{attribute addProperty BoxType "EP7342-0002-0021"}
{attribute addProperty Id "ENC_Status_compact_ChannelAT %I*ARRAY[0..1] OF ENC_Status_compact_Channel_A7E8355C96120DCM_Status_ChannelAT %I*ARRAY[0..1] OF DCM_Status_Channel_64D937433240ENC_Control_compact_ChannelAT %Q*ARRAY[0..1] OF ENC_Control_compact_Channel_5C86AA9D6480DCM_Control_Channel_1AT %Q*DCM_Control_Channel_6F24B2C41620DCM_Velocity_Channel_1AT %Q*DCM_Velocity_Channel_1D89B5C21620DCM_Control_Channel_2AT %Q*DCM_Control_Channel_6F24B2C41620DCM_Velocity_Channel_2AT %Q*DCM_Velocity_Channel_1D89B5C21620WcStateAT %I*WcState_F855686C1620InfoDataAT %I*InfoData_3F3BB279112140"}
{attribute addProperty CRC "3653863044"}
{attribute addProperty SizeInBites "384"}
{attribute addProperty SizeInBytes "48"}
TYPE EP7342_014E0448 :
STRUCT
	{attribute addProperty Name "ENC_Status_compact_Channel"}
	ENC_Status_compact_Channel : ARRAY[0..1] OF ENC_Status_compact_Channel_A7E8355C;
	{attribute addProperty Name "DCM_Status_Channel"}
	DCM_Status_Channel : ARRAY[0..1] OF DCM_Status_Channel_64D93743;
	{attribute addProperty Name "ENC_Control_compact_Channel"}
	ENC_Control_compact_Channel : ARRAY[0..1] OF ENC_Control_compact_Channel_5C86AA9D;
	{attribute addProperty Name "DCM_Control_Channel_1"}
	DCM_Control_Channel_1 : DCM_Control_Channel_6F24B2C4;
	{attribute addProperty Name "DCM_Velocity_Channel_1"}
	DCM_Velocity_Channel_1 : DCM_Velocity_Channel_1D89B5C2;
	{attribute addProperty Name "DCM_Control_Channel_2"}
	DCM_Control_Channel_2 : DCM_Control_Channel_6F24B2C4;
	{attribute addProperty Name "DCM_Velocity_Channel_2"}
	DCM_Velocity_Channel_2 : DCM_Velocity_Channel_1D89B5C2;
	{attribute addProperty Name "WcState"}
	WcState : WcState_F855686C;
	{attribute addProperty Name "InfoData"}
	InfoData : InfoData_3F3BB279;
END_STRUCT
END_TYPE

(* stored: Version 1.2.0.0, ProductVersion 3.1.4024.9
   DUT EP7342_014E0448: Id {9857c686-dd88-429d-ba88-f4791d64d0fc} *)
